DATA_BLOCK "EM_Rotator_Pendant_DB"
{ S7_Optimized_Access := 'TRUE' }
VERSION : 0.1
"EM_Rotator_Pendant"
BEGIN
END_DATA_BLOCK
